(*$
	Returns <i>TRUE</i> if the status of the instance <b><i>this</i></b> is
	<a href="#jog_manager_status_enum"><i>JOG_MANAGER_STATUS_ACTIVE</i></a>
	and  <i>list_selected</i> is a valid index,
	<i>FALSE</i> otherwise.
$*)
FUNCTION jog_manager_is_jog_axis_deactivating : BOOL
VAR_INPUT
	index:				UINT;
END_VAR
VAR_IN_OUT
    CONVERSION_this:	jog_manager;	(*$ Instance to which the method applies $*)
END_VAR

IF	(
		(CONVERSION_this.CONVERSION_private.list_selected <> CONVERSION_this.CONVERSION_private.old_list_selected)
		OR
		(CONVERSION_this.status = JOG_MANAGER_STATUS_SEL_DISABLE_AXIS)		
	)
	AND
	(CONVERSION_this.CONVERSION_private.old_list_selected = index)
	AND	
	CONVERSION_this.CONVERSION_private.old_list_selected_axis_is_valid
THEN
	jog_manager_is_jog_axis_deactivating := (CONVERSION_this.status >= JOG_MANAGER_STATUS_ACTIVE);
ELSE
	jog_manager_is_jog_axis_deactivating := FALSE;
END_IF

END_FUNCTION

(* stored: Version 1.1.0.1, ProductVersion 3.1.4022.12
   POU jog_manager_is_jog_axis_deactivating: Id {b0e0c804-8061-4eb9-86c8-ba84ed921d55}, SpecialFunc None *)
